Omron CX-Programmer project NewProject (CX-Programmer 9.51)

# PLC my_first_project: CP1L L
; MyfirstProject

## Global symbols (name address type ; comment)
T0001 BOOL  ; Timer number

## Program NewProgram1 (cyclic task 0)
Local symbols
TOOO1 0.05 BOOL
TOOOO 0.04 BOOL
button_1 0.00 BOOL
out_2 100.01 BOOL

### Section Section1

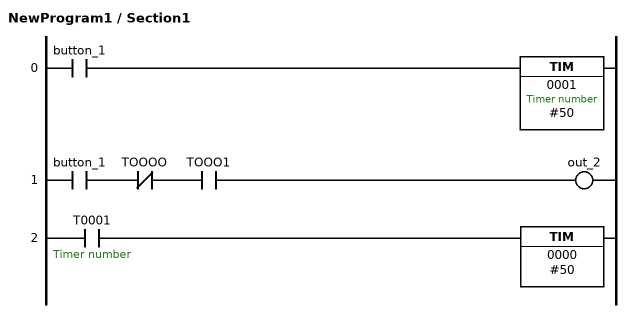
; rung 0
LD button_1
TIM 0001 #50  ; Timer number
; rung 1
LD button_1
ANDNOT TOOOO
AND TOOO1
OUT out_2
; rung 2
LD T0001  ; Timer number
TIM 0000 #50

### Section END
; rung 0
END(001)